FUNCTION_BLOCK JsonLinkSettingsParser IMPLEMENTS I_LinkSettings
VAR
	parser : REFERENCE TO FB_JsonDomParser;
	baseJsonValue : SJsonValue;
	jsonLanguagePack : I_JsonLanguagePack;
END_VAR

PROPERTY PUBLIC DestinationId : NodeId
GET
VAR
	jsonValue: SJsonValue;
END_VAR
VAR CONSTANT
	DESTINATION_ID_POS : UDINT := 3;
END_VAR
jsonValue := parser.GetArrayValueByIdx(baseJsonValue, DESTINATION_ID_POS);
DestinationId := DINT_TO_INT(parser.GetInt(jsonValue));
END_GET
END_PROPERTY

PROPERTY PUBLIC DestinationPortId : PortId
GET
VAR
	jsonValue: SJsonValue;
END_VAR
VAR CONSTANT
	DESTINATION_PORT_ID_POS : UDINT := 4;
END_VAR
jsonValue := parser.GetArrayValueByIdx(baseJsonValue, DESTINATION_PORT_ID_POS);
DestinationPortId := DINT_TO_INT(parser.GetInt(jsonValue));
END_GET
END_PROPERTY

METHOD FB_init : BOOL
VAR_INPUT
	bInitRetains : BOOL; // if TRUE, the retain variables are initialized (warm start / cold start)
	bInCopyCode : BOOL;  // if TRUE, the instance afterwards gets moved into the copy code (online change)
	JsonLanguagePack : I_JsonLanguagePack;
END_VAR
THIS^.jsonLanguagePack := JsonLanguagePack;
END_METHOD

PROPERTY PUBLIC Id : T_MAXSTRING
GET
VAR
	jsonValue: SJsonValue;
END_VAR
VAR CONSTANT
	ID_POS : UDINT := 0;
END_VAR
jsonValue := parser.GetArrayValueByIdx(baseJsonValue, ID_POS);
Id := DINT_TO_STRING(parser.GetInt(jsonValue));
END_GET
END_PROPERTY

PROPERTY PUBLIC SourceId : NodeId
GET
VAR
	jsonValue: SJsonValue;
END_VAR
VAR CONSTANT
	SOURCE_ID_POS : UDINT := 1;
END_VAR
jsonValue := parser.GetArrayValueByIdx(baseJsonValue, SOURCE_ID_POS);
SourceId := DINT_TO_INT(parser.GetInt(jsonValue));
END_GET
END_PROPERTY

PROPERTY PUBLIC SourcePortId : PortId
GET
VAR
	jsonValue: SJsonValue;
END_VAR
VAR CONSTANT
	SOURCE_PORT_ID_POS : UDINT := 2;
END_VAR
jsonValue := parser.GetArrayValueByIdx(baseJsonValue, SOURCE_PORT_ID_POS);
SourcePortId := DINT_TO_INT(parser.GetInt(jsonValue));
END_GET
END_PROPERTY

METHOD PUBLIC Update
VAR_INPUT
	Parser : REFERENCE TO FB_JsonDomParser;
	JsonValue : SJsonValue;
END_VAR
THIS^.parser REF= Parser;
THIS^.baseJsonValue := JsonValue;
END_METHOD

END_FUNCTION_BLOCK

(* stored: Version 1.1.0.1, ProductVersion 3.1.4024.12
   POU JsonLinkSettingsParser: Id {34e63be9-68fb-00e6-1a36-e868df41ef3c}, SpecialFunc None
   Folder Constructor: Id {752d120f-7241-031b-390a-b086a9c42882}
   Property DestinationId: Id {06b6421d-1335-0ecd-1f75-c3899581f456}
   Get Get: Id {20562751-4ae4-091d-2ecc-16e1ce1b1e74}
   Property DestinationPortId: Id {ba9eb1fc-0ac2-098f-3e85-67e7b4294ee8}
   Get Get: Id {9b2d2cf8-90d9-097e-0682-166168729700}
   Method FB_init: Id {02aab07c-d105-00bb-3c30-57aee63d2afe}
   Property Id: Id {107931e8-48a8-089e-25df-5902f7d2b943}
   Get Get: Id {d0a394b5-3a46-0d4b-24f4-98e46377d2c3}
   Property SourceId: Id {4dfb2bd7-5e35-0fae-1b13-53e945558fb6}
   Get Get: Id {97760a9e-c7e3-0e8f-253e-6b96f4db32d4}
   Property SourcePortId: Id {e8d9aead-996f-0ff6-3d80-3abf21b78b49}
   Get Get: Id {612d3d99-4ee9-00ac-1180-b9981362633a}
   Method Update: Id {caf16119-5d16-04ed-0212-e5fe8f438e71} *)
